// TIA Portal V20 export
ORGANIZATION_BLOCK "Main"   // OB126, LAD, ProgramCycle
TITLE = "Main Program Sweep (Cycle)"
// stored: Namespace CITI_Logic, SetENOAutomatically false
   VAR_INPUT
      Initial_Call : Bool;   // Initial call of this OB
      Remanence : Bool;   // =True, if remanent data are available
   END_VAR
BEGIN

REGION Network 1: PMC_Map00
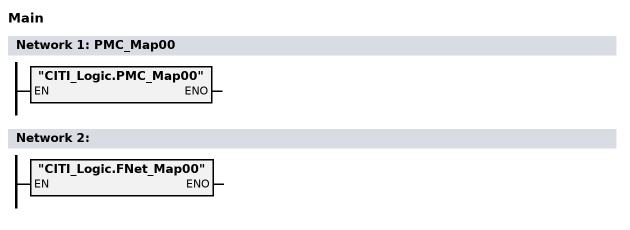
   RUNG wire#powerrail
      "CITI_Logic.PMC_Map00"()
   END_RUNG
   // the same network as SCL:
   "CITI_Logic.PMC_Map00"();
END_REGION

REGION Network 2
   RUNG wire#powerrail
      "CITI_Logic.FNet_Map00"()
   END_RUNG
   // the same network as SCL:
   "CITI_Logic.FNet_Map00"();
END_REGION
END_ORGANIZATION_BLOCK
